FUNCTION F_WindowColor (* Pick u8ColorIn if rValue lies within [rMin, rMax], otherwise u8ColorOut. *)
  (* Standard: 61499-2; Description: Copyright (c) 2026 Meisterschulen am Ostbahnhof This program and the accompanying materials are made available under the terms of the Eclipse Public License 2.0 which is available at https://www.eclipse.org/legal/epl-2.0/ SPDX-License-Identifier: EPL-2.0 *)
  (* Version 1.0, 2026-09-06, Franz Höpfinger, Meisterschulen am Ostbahnhof, initial API and implementation and/or initial documentation *)
  PACKAGE isobus::UT::Q::helpers;
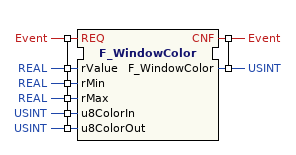
  EVENT_INPUT
    REQ WITH rValue, rMin, rMax, u8ColorIn, u8ColorOut;
  END_EVENT
  EVENT_OUTPUT
    CNF WITH F_WindowColor;
  END_EVENT
  VAR_INPUT
    rValue : REAL;
    rMin : REAL;
    rMax : REAL;
    u8ColorIn : USINT; (* Returned when rMin <= rValue <= rMax *)
    u8ColorOut : USINT; (* Returned otherwise *)
  END_VAR
  VAR_OUTPUT
    F_WindowColor : USINT;
  END_VAR
  BODY IN ST:
PACKAGE isobus::UT::Q::helpers;

(* Pick u8ColorIn if rValue lies within [rMin, rMax], otherwise u8ColorOut. *)
FUNCTION F_WindowColor : USINT

VAR_INPUT
	rValue : REAL;
	rMin : REAL;
	rMax : REAL;
	u8ColorIn : USINT;
	u8ColorOut : USINT;
END_VAR

IF rValue >= rMin AND rValue <= rMax THEN
	F_WindowColor := u8ColorIn;
ELSE
	F_WindowColor := u8ColorOut;
END_IF;

END_FUNCTION
  END_BODY
END_FUNCTION
